FUNCTION_BLOCK Q_NumericValue_AUDI (* Command change numeric value ( Part 6 - F.22 ) *)
  (* Standard: ISO 11783-6; Description: Copyright (c) 2022 HR Agrartechnik GmbH This program and the accompanying materials are made available under the terms of the Eclipse Public License 2.0 which is available at https://www.eclipse.org/legal/epl-2.0/ SPDX-License-Identifier: EPL-2.0 see Description Tab *)
  (* Version 1.0, 2022-07-08, Franz Höpfinger, HR Agrartechnik GmbH *)
  PACKAGE isobus::UT::Q;
  IMPORT eclipse4diac::core::TypeHash;
  IMPORT isobus::UT::Q::const::IDs::ID_NULL;
  (* Documentation:
  Command change numeric value ( Part 6 - F.22 )
   This command is used to change the value of an object. It applies only to objects that have a numeric value attribute.
   param[in] {objectID, uint16_t}
   Object ID
   param[in] {value, uint32_t}
   New value of ID
   Return Values: 
   int16_t
    - VT_E_NO_ERR (0) - OK
   - VT_E_OVERFLOW (-6) - buffer overflow
   - VT_E_NOACT (-8) - Command not possible in current state
   - VT_E_NO_INSTANCE (-21) - No VT client available
   - VT_E_ISO_INSTANCE_INVALID (-129) - Identifier for instance (connection) invalid
   - VT_E_HANDLE_INVALID (-128) - ErrorCause: invalid Handle
   - VT_E_NOT_ALIVE (-130) - Identifier for instance valid, but VT Dead.
  *)
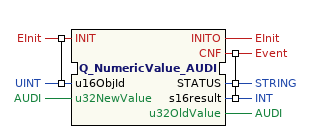
  EVENT_INPUT
    INIT : EInit WITH u16ObjId; (* Service Initialization *)
  END_EVENT
  EVENT_OUTPUT
    INITO : EInit; (* Initialization Confirm *)
    CNF WITH STATUS, s16result; (* Confirmation of Requested Service *)
  END_EVENT
  VAR_INPUT
    u16ObjId : UINT := ID_NULL; (* Object ID *)
  END_VAR
  VAR_OUTPUT
    STATUS : STRING; (* Service Status *)
    s16result : INT; (* retval see description *)
  END_VAR
  SOCKETS
    u32NewValue : adapter::types::unidirectional::AUDI; (* New value of ID *)
  END_SOCKETS
  PLUGS
    u32OldValue : adapter::types::unidirectional::AUDI; (* Old value of ID *)
  END_PLUGS
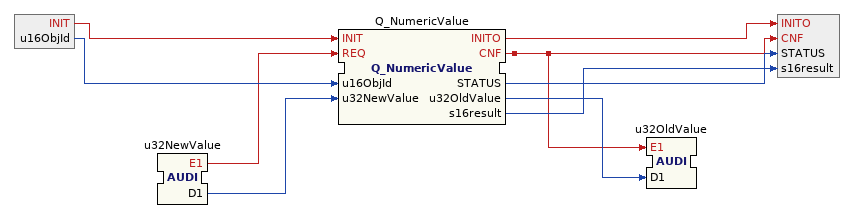
  FBS
    Q_NumericValue : isobus::UT::Q::Q_NumericValue;
  END_FBS
  EVENT_CONNECTIONS
    INIT TO Q_NumericValue.INIT;
    Q_NumericValue.INITO TO INITO;
    Q_NumericValue.CNF TO CNF;
    u32NewValue.E1 TO Q_NumericValue.REQ;
    Q_NumericValue.CNF TO u32OldValue.E1;
  END_CONNECTIONS
  DATA_CONNECTIONS
    Q_NumericValue.STATUS TO STATUS;
    u16ObjId TO Q_NumericValue.u16ObjId;
    u32NewValue.D1 TO Q_NumericValue.u32NewValue;
    Q_NumericValue.u32OldValue TO u32OldValue.D1;
    Q_NumericValue.s16result TO s16result;
  END_CONNECTIONS
END_FUNCTION_BLOCK
